{attribute 'no_explicit_call' := 'Do not call this POU directly'}
FUNCTION_BLOCK LiftManager

VAR
	_myLiftActuator : ITF_LiftActuator;
	
	iState: INT;
END_VAR

METHOD Cycle : BOOL
VAR_INPUT
END_VAR
CASE iState OF 	

	1:
		_myLiftActuator.ExtendActuator();
		iState := 0;
	2:
		_myLiftActuator.RetractActuator();
		iState := 0;
END_CASE
END_METHOD

PROPERTY MyLiftActuator : ITF_LiftActuator
GET
END_GET
SET
END_SET
END_PROPERTY

END_FUNCTION_BLOCK

(* stored: Version 1.1.0.1
   POU LiftManager: Id {b519674b-042e-4629-a2ce-f61971732cfa}, SpecialFunc None
   Method Cycle: Id {15ed8f4f-1b4c-47be-8e57-2db6c6c259e2}
   Property MyLiftActuator: Id {84577b43-26ad-4a3b-b509-ed180b27bc1e}
   Get Get: Id {c0262f38-7bad-4343-ba8b-3345bfffab51}
   Set Set: Id {d232a965-229a-477d-a70e-138a856406d8} *)
